(* PLC project Tc2_Utilities.FindAndDelete Demo, tc3-libraries-kb TwinCAT 3.1 *)
(* stored: creationDateTime 2026-05-10T16:00:00, modificationDateTime 2026-05-10T16:00:00 *)

PROGRAM P_Demo_FindAndDelete
  VAR
    rResult : UDINT;  (* FindAndDelete 返回值 *)
    bRun : BOOL;  (* 触发一次调用 *)
    sIn : STRING(255) := 'foo bar foo baz foo';  (* 测试用本地变量 *)
    sDel : STRING(31) := 'foo';  (* 测试用本地变量 *)
    sOut : STRING(255);  (* 测试用本地变量 *)
  END_VAR

            // ============================================================
// Tc2_Utilities.FindAndDelete 演示程序（FUNCTION）
// ============================================================
// 验证步骤：
//   1. 引用 Tc2_Utilities
//   2. 编译 + 登录
//   3. 强制 bRun := TRUE 一个周期
//   4. 在线监视 rResult / 各 demo 变量
// ============================================================

IF bRun THEN
    rResult := FindAndDelete(ADR(sIn), ADR(sDel), ADR(sOut), SIZEOF(sOut));
    bRun := FALSE;
END_IF;

          
END_PROGRAM
